VAR_GLOBAL CONSTANT
    gcMaxLVC4000	:	INT := 20; //maximum number of LVC4000 units per port
END_VAR

(* stored: Version 1.1.0.1
   GVL GVL_MacroSensorsParameters: Id {1082d9c1-a21d-43e2-a315-2445bcd762d2} *)
